FUNCTION_BLOCK LINE (* openCV line drawer *)
  (* Version 1.0, AN, SWDC RTSoft *)
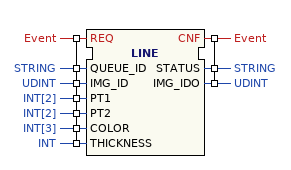
  EVENT_INPUT
    REQ WITH QUEUE_ID, IMG_ID, PT1, PT2, COLOR, THICKNESS;
  END_EVENT
  EVENT_OUTPUT
    CNF WITH STATUS, IMG_IDO;
  END_EVENT
  VAR_INPUT
    QUEUE_ID : STRING;
    IMG_ID : UDINT;
    PT1 : ARRAY [0..1] OF INT; (* Start point of the line [x, y] *)
    PT2 : ARRAY [0..1] OF INT; (* End point of the line [x, y] *)
    COLOR : ARRAY [0..2] OF INT; (* [B, G, R] *)
    THICKNESS : INT;
  END_VAR
  VAR_OUTPUT
    STATUS : STRING;
    IMG_IDO : UDINT;
  END_VAR
  ALGORITHM REQ IN ST:

  END_ALGORITHM
END_FUNCTION_BLOCK
